{attribute 'linkalways'} 
{attribute 'no_explicit_call' := 'This FB is a CLASS and must be accessed using methods or properties'}
{attribute 'enable_dynamic_creation'}
FUNCTION_BLOCK IncorrectTypeDeserializationError EXTENDS Error
VAR
	dataType : T_MAXSTRING;
END_VAR

PROPERTY PUBLIC ErrorType : T_MAXSTRING
GET
ErrorType := 'INCORRECT_DATATYPE_DESERIALIZATION_ERROR';
END_GET
END_PROPERTY

METHOD FB_init : BOOL
VAR_INPUT
	bInitRetains : BOOL; // if TRUE, the retain variables are initialized (warm start / cold start)
	bInCopyCode : BOOL;  // if TRUE, the instance afterwards gets moved into the copy code (online change)
	DataType : T_MAXSTRING;
END_VAR
THIS^.dataType := DataType;
END_METHOD

PROPERTY PUBLIC Message : T_MAXSTRING
GET
Message := CONCAT('Deserialization Failed, Incorrect Datatype : ', dataType);
END_GET
END_PROPERTY

END_FUNCTION_BLOCK

(* stored: Version 1.1.0.1, ProductVersion 3.1.4024.12
   POU IncorrectTypeDeserializationError: Id {0000e4f8-94a9-07e8-1199-197adeaa849d}, SpecialFunc None
   Folder Constructor: Id {70744e12-2266-04d6-1157-7243aa266801}
   Property ErrorType: Id {46abd7d5-fddd-0a0b-2254-63a77b02d0ff}
   Get Get: Id {25bd366e-ebc9-089d-27a0-a90e208ae939}
   Method FB_init: Id {1add5e11-dd8f-0c5a-1c68-26bca88bbd84}
   Property Message: Id {8f377fc1-f2f7-0c33-0568-e1ddd548eca5}
   Get Get: Id {17f0e272-a7a4-016a-0b96-ef3ad78e0401} *)
